INTERFACE I_PackML_HoldingCommands

METHOD PUBLIC Abort
VAR_INPUT
END_VAR
END_METHOD

METHOD StateComplete
VAR_INPUT
END_VAR
END_METHOD

METHOD PUBLIC Stop
VAR_INPUT
END_VAR
END_METHOD

END_INTERFACE

(* stored: Version 1.1.0.1, ProductVersion 3.1.4024.12
   Itf I_PackML_HoldingCommands: Id {af08fee2-ed8e-0073-1bb5-3408d155c093}
   Method Abort: Id {6e242917-794f-06a0-21b8-fe2adc554005}
   Method StateComplete: Id {bdf98d5c-18e8-0cc0-2fd2-68ee2dd7f5f4}
   Method Stop: Id {07ea8dc0-579c-0129-26da-243e5eb95edf} *)
